TYPE ST_Signals :
STRUCT
	fOutSignal 				: LREAL; // Signal Sent Out
	fOutCompansated			: LREAL; // DB Compansated, NOT IN USE
	fFF						: LREAL; // FeedForward Signal
	fPID					: LREAL; // PID Signal
	fError					: LREAL; // Signal Error
	fU						: LREAL; // FF + PID + DB
	fUAdj					: LREAL; // Adjusted U, for flow sharing
END_STRUCT
END_TYPE

(* stored: Version 1.1.0.1
   DUT ST_Signals: Id {1a8d1cb5-ae4d-41a6-919c-e179c49138cd} *)
